PROGRAM P_Robot_Operate
VAR
END_VAR

//No implements

END_PROGRAM

(* stored: Version 1.1.0.1, ProductVersion 3.1.4024.15
   POU P_Robot_Operate: Id {d6914ce3-ccac-49af-81dd-d937c420ed91}, SpecialFunc None *)
